FUNCTION_BLOCK REAL_MIN (* Basic Function Block Type *)
  (* Standard: 61499-2 *)
  (* Version 0.0, 1/27/2023, brink, Flexbridge AB, Template *)
  PACKAGE UAO.Hackathon;
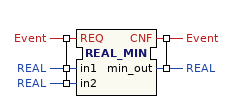
  EVENT_INPUT
    REQ WITH in1, in2; (* Normal Execution Request *)
  END_EVENT
  EVENT_OUTPUT
    CNF WITH min_out; (* Execution Confirmation *)
  END_EVENT
  VAR_INPUT
    in1 : REAL; (* Input event qualifier *)
    in2 : REAL;
  END_VAR
  VAR_OUTPUT
    min_out : REAL; (* Output event qualifier *)
  END_VAR
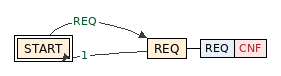
  EC_STATES
    START; (* Initial State *)
    REQ : REQ -> CNF; (* Normal execution *)
  END_STATES
  EC_TRANSITIONS
    START TO REQ := REQ;
    REQ TO START := 1;
  END_TRANSITIONS
  ALGORITHM REQ IN ST: (* Normally executed algorithm *)
min_out := MIN(in1, in2);
  END_ALGORITHM
END_FUNCTION_BLOCK
